FUNCTION UpdateEventTimestampWithSystemTime
VAR_INPUT
	stEvent : REFERENCE TO ST_Event;
END_VAR
VAR
	fbGETSYSTEMTIME : GETSYSTEMTIME;
	stFileName : T_FILETIME;
END_VAR

fbGETSYSTEMTIME(timeLoDW=>stFileName.dwLowDateTime,
 timeHiDW => stFileName.dwHighDateTime);
 
stEvent.dtTimeStamp := FILETIME_TO_DT(fileTime := stFileName);

END_FUNCTION

(* stored: Version 1.1.0.1, ProductVersion 3.1.4024.12
   POU UpdateEventTimestampWithSystemTime: Id {e7770d6b-193e-4a84-a69e-4e1b60ba3725}, SpecialFunc None *)
